FUNCTION_BLOCK X20DI9371 (* Digital inputs at the openPOWERLINK fieldbus *)
  (* Standard: 61499-2; Description: Copyright (c) 2011 AIT This program and the accompanying materials are made available under the terms of the Eclipse Public License 2.0 which is available at https://www.eclipse.org/legal/epl-2.0/ SPDX-License-Identifier: EPL-2.0 *)
  (* Version 0.0, 2011-05-31, Filip Andren, AIT *)
  (* Version 1.0, 2011-05-31, Filip Andren, Thomas Strasser, AIT *)
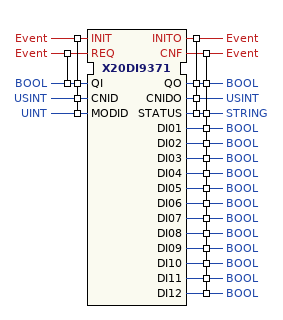
  EVENT_INPUT
    INIT WITH QI, CNID, MODID; (* Service Initialization *)
    REQ WITH QI; (* Application Response to IND *)
  END_EVENT
  EVENT_OUTPUT
    INITO WITH QO, STATUS, CNIDO; (* Initialization Confirm *)
    CNF WITH DI01, DI02, DI03, DI04, DI05, DI06, DI07, DI08, DI09, DI10, DI11, DI12, STATUS, QO; (* Indication from Resource *)
  END_EVENT
  VAR_INPUT
    QI : BOOL; (* Event Input Qualifier *)
    CNID : USINT; (* Client Node ID *)
    MODID : UINT; (* Station Number *)
  END_VAR
  VAR_OUTPUT
    QO : BOOL; (* Event Output Qualifier *)
    CNIDO : USINT; (* Client Node ID Output *)
    STATUS : STRING; (* Service Status *)
    DI01 : BOOL; (* Digital Input 01 *)
    DI02 : BOOL; (* Digital Input 02 *)
    DI03 : BOOL; (* Digital Input 03 *)
    DI04 : BOOL; (* Digital Input 04 *)
    DI05 : BOOL; (* Digital Input 05 *)
    DI06 : BOOL; (* Digital Input 06 *)
    DI07 : BOOL; (* Digital Input 07 *)
    DI08 : BOOL; (* Digital Input 08 *)
    DI09 : BOOL; (* Digital Input 09 *)
    DI10 : BOOL; (* Digital Input 10 *)
    DI11 : BOOL; (* Digital Input 11 *)
    DI12 : BOOL; (* Digital Input 12 *)
  END_VAR
  SERVICE APPLICATION/RESOURCE (* Service Interface Function Block Type *)
    SEQUENCE normal_establishment
      APPLICATION.INIT+(PARAMS) -> APPLICATION.INITO+(PARAMS);
    END_SEQUENCE
    SEQUENCE unsuccessful_establishment
      APPLICATION.INIT+(PARAMS) -> APPLICATION.INITO-(STATUS);
    END_SEQUENCE
    SEQUENCE request_confirm
      APPLICATION.REQ+(SD) -> APPLICATION.CNF+(RD);
    END_SEQUENCE
    SEQUENCE request_inhibited
      APPLICATION.REQ-(SD) -> APPLICATION.CNF-(STATUS);
    END_SEQUENCE
    SEQUENCE request_error
      APPLICATION.REQ+(SD) -> APPLICATION.CNF-(STATUS);
    END_SEQUENCE
    SEQUENCE indication_response
      RESOURCE.indicate(RD) -> APPLICATION.IND+(RD);
      APPLICATION.RSP(QI,SD) -> RESOURCE.response(QI,SD);
    END_SEQUENCE
    SEQUENCE indication_inhibited
      RESOURCE.indicate(RD,QI=FALSE) -> RESOURCE.inhibited();
    END_SEQUENCE
    SEQUENCE error_indication
      RESOURCE.error(STATUS) -> APPLICATION.IND-(STATUS);
    END_SEQUENCE
    SEQUENCE application_initiated_termination
      APPLICATION.INIT-() -> APPLICATION.INITO-(STATUS);
    END_SEQUENCE
    SEQUENCE resource_initiated_termination
      -> APPLICATION.INITO-(STATUS);
    END_SEQUENCE
  END_SERVICE
END_FUNCTION_BLOCK
